(* CODESYS project Uppgift 9.project

Project tree, tasks and I/O mapping:
  Device : CODESYS Control Win V3, 3S - Smart Software Solutions GmbH, order no. 305021, version 3.5.10.40
    application Application
      libraries: Standard, * (System)
      task MainTask (cyclic, interval t#20ms, priority 1) calls PLC_PRG
      task VISU_TASK (cyclic, interval 100 ms, priority 31) calls VisuElems.Visu_Prg
      program PLC_PRG [LD]
      visualisation Visualization
  libraries: VisuSymbols, 3.5.10.0 (System)
  text list GlobalTextList
*)

// Device/Application/PLC_PRG
PROGRAM PLC_PRG
VAR
	TON_0: TON;
	Green_Lamp: BOOL;
	Blue_Lamp: BOOL;
	Yellow_Lamp: BOOL;
	Btn_1: BOOL;
	Timeoutput: TIME;
	TOF_0: TOF;
	TOF_1: TOF;
	TOF_2: TOF;
	Returnvalue: BOOL;
	BluLampCounter: TIME;
	YellowLampCounter: TIME;
	ReturnvaluCounter: TIME;
	TOF_1gdf: TOn;
	TOF_0df: TOn;
	TOF_2df: TOn;
	TP_0: TP;
	Btn_1_output: BOOL;
END_VAR

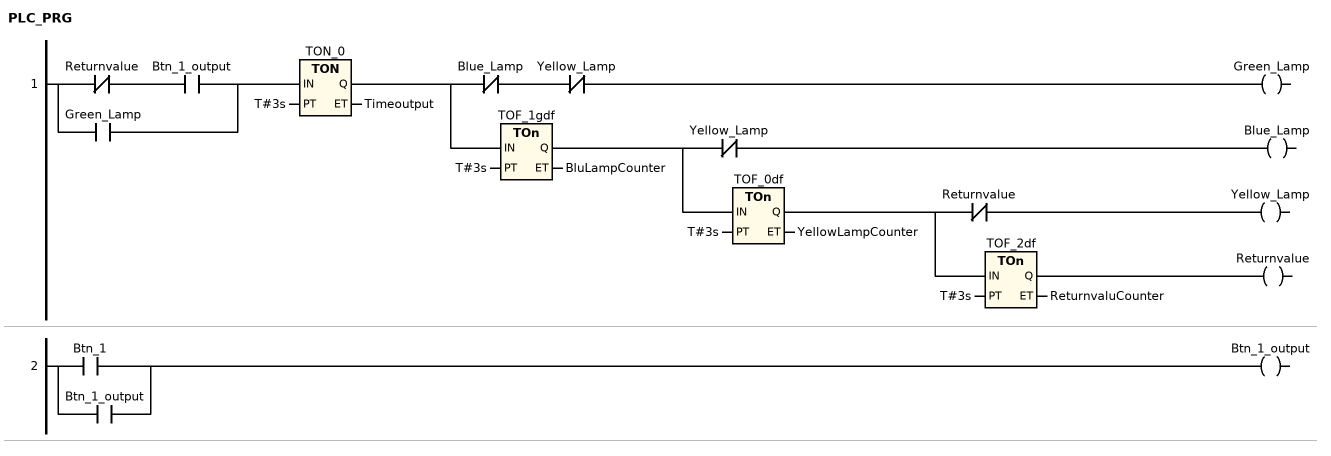
// NETWORK 1
TON_0(IN := NOT Returnvalue AND Btn_1_output OR Green_Lamp, PT := T#3s, ET => Timeoutput); // TON
Green_Lamp := TON_0.Q AND NOT Blue_Lamp AND NOT Yellow_Lamp;
TOF_1gdf(IN := TON_0.Q, PT := T#3s, ET => BluLampCounter); // TOn
Blue_Lamp := TOF_1gdf.Q AND NOT Yellow_Lamp;
TOF_0df(IN := TOF_1gdf.Q, PT := T#3s, ET => YellowLampCounter); // TOn
Yellow_Lamp := TOF_0df.Q AND NOT Returnvalue;
TOF_2df(IN := TOF_0df.Q, PT := T#3s, ET => ReturnvaluCounter); // TOn
Returnvalue := TOF_2df.Q;

// NETWORK 2
Btn_1_output := Btn_1 OR Btn_1_output;

END_PROGRAM

// Device/Application/Visualization
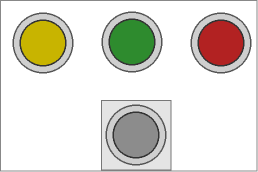
VISUALIZATION Visualization  // 258x172
    Lamp1 (8,8 70x70), style: Lamp-Lamp1-Yellow
    Lamp1 (97,7 70x70), style: Lamp-Lamp1-Green
    Lamp1 (186,8 70x70), style: Lamp-Lamp1-Red
    PushSwitch (101,100 70x70), behaviour: TOGGLE, style: Switch-PushSwitch-Gray
END_VISUALIZATION
